(* PLC project LadderFidelityFixture, greenforge-labs codescribe-fixture 1 *)
(* stored: creationDateTime 2020-01-01T00:00:00 *)

PROGRAM LD_FIDELITY
  VAR
    xGo : BOOL;
    xStart : BOOL;
    xManual : BOOL;
    xDone : BOOL;
    iCount : INT;
    ctr : CTU;
    xPress : BOOL;
    xStop : BOOL;
    xRun : BOOL;
    xCool : BOOL;
    tmr2 : TON;
    xB : BOOL;
    xGo2 : BOOL;
    xFin : BOOL;
    tmrA : TON;
    ctr2 : CTU;
    tmrD : TON;
  END_VAR

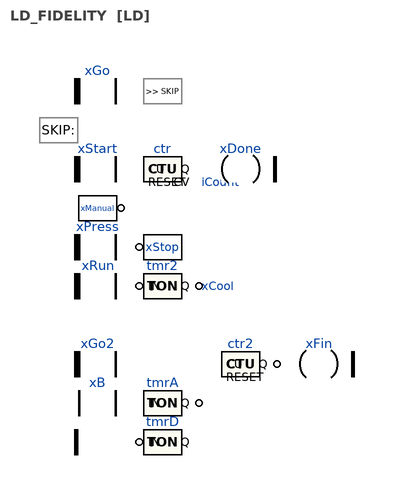
(* LD diagram, written out as Structured Text *)
IF xGo THEN JMP SKIP; END_IF;
SKIP:
ctr(CU := xStart, RESET := NOT xManual, CV => iCount);
xDone := ctr.Q;
xStop := NOT xPress;
tmrA(IN := xB);
ctr2(CU := xGo2, RESET := NOT tmrA.Q);
xFin := NOT ctr2.Q;
tmr2(IN := NOT xRun, Q => xCool);
tmrD(IN := NOT TRUE);
END_PROGRAM
